// TIA Portal V17 export
// export: Created 2025-03-07T09:19:12.5870165Z, ExportSetting WithDefaults, DisplayName Totally Integrated Automation Portal, DisplayVersion V17 Update 8, DisplayName TIA Portal Openness, DisplayVersion V17 Update 8, DisplayName TIA Portal Version Control Interface, DisplayVersion V17, DisplayName SINAMICS Startdrive Advanced, DisplayVersion V17 SP2, DisplayName SINAMICS Startdrive G110M, G120, G120C, G120D, G120P, G115D, DisplayVersion V17 SP2, DisplayName SINAMICS Startdrive G130, G150, S120, S150, SINAMICS MV, S210, DisplayVersion V17 SP2, DisplayName STEP 7 Professional, DisplayVersion V17 Update 8, DisplayName SINUMERIK ONE STEP 7 Toolbox, DisplayVersion V17 Update 12, DisplayName SINUMERIK 840D sl STEP 7 Toolbox, DisplayVersion V17 Update 12, DisplayName STEP 7 Safety, DisplayVersion V17 Update 6, DisplayName WinCC Advanced, DisplayVersion V17 Update 8
FUNCTION "FC7210_PRODUCTION" : Void   // FC7210, LAD
{ S7_Optimized_Access := 'FALSE' }
AUTHOR : ETXETAR
VERSION : 1.0
// stored: AutoNumber false, IsIECCheckEnabled false, SetENOAutomatically false, UDAEnableTagReadback false
   VAR_TEMP
      UNIT_01_ENABLE_COUNT : Bool;   // UNIT 01 ENABLE COUNT
      UNIT_02_ENABLE_COUNT : Bool;   // UNIT 02 ENABLE COUNT
   END_VAR
   VAR_TEMP   // added for the SCL form of the ladder/FBD networks
      _w1 : Bool;
   END_VAR
BEGIN

REGION Network 1: UNIT 01 ENABLE COUNT / ENABLE FIXTURE 1 COUNT
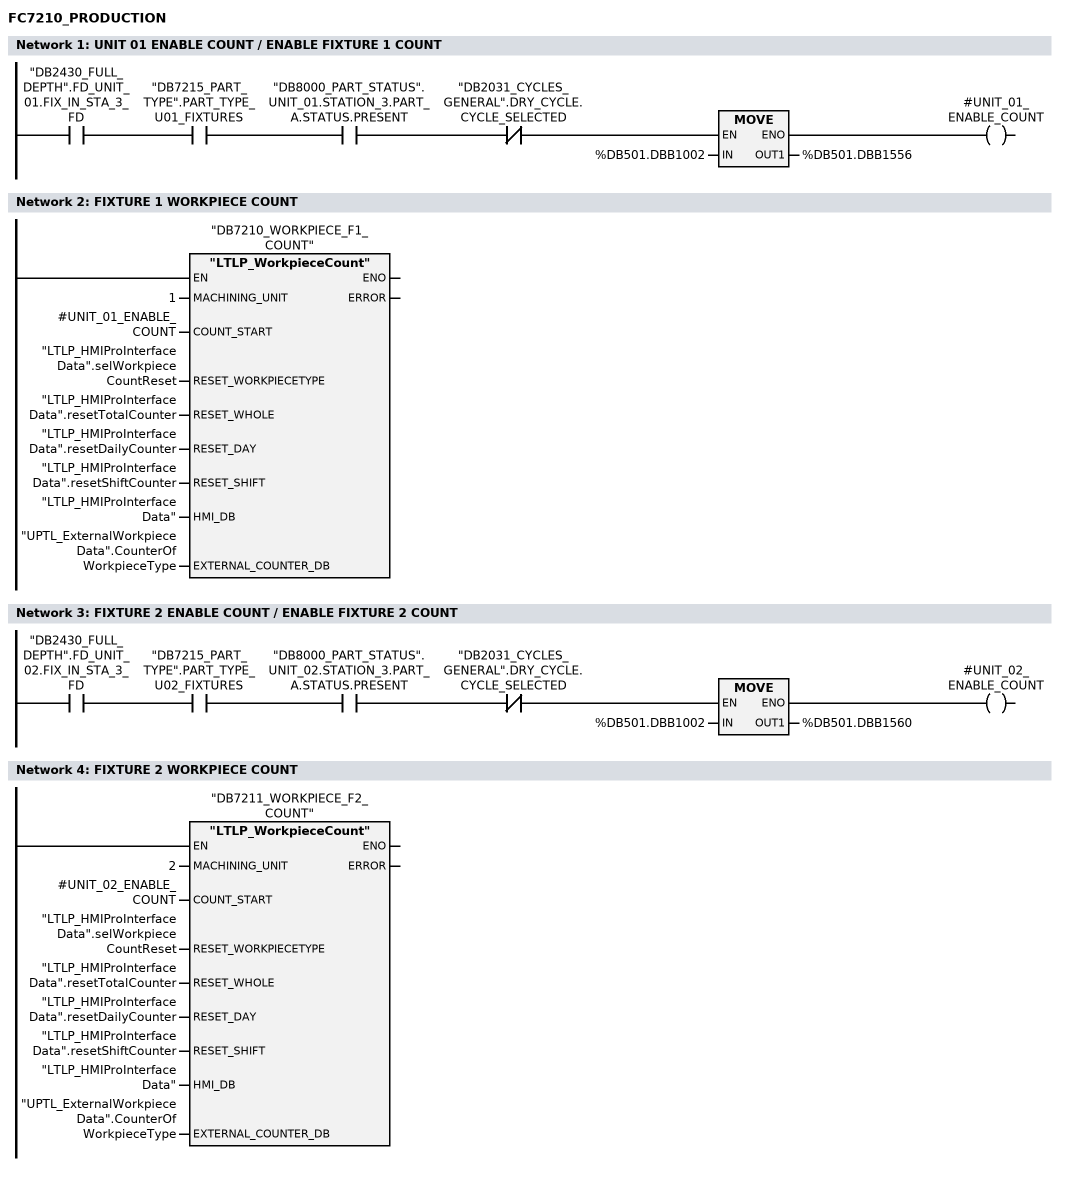
   RUNG wire#powerrail
      Contact( "DB2430_FULL_DEPTH".FD_UNIT_01.FIX_IN_STA_3_FD )
      Contact( "DB7215_PART_TYPE".PART_TYPE_U01_FIXTURES )
      Contact( "DB8000_PART_STATUS".UNIT_01.STATION_3.PART_A.STATUS.PRESENT )
      I_Contact( "DB2031_CYCLES_GENERAL".DRY_CYCLE.CYCLE_SELECTED )
      Move(in := %DB501.DBB1002, out1 => %DB501.DBB1556)
      Coil( #UNIT_01_ENABLE_COUNT )
   END_RUNG
   // the same network as SCL:
   #_w1 := "DB2430_FULL_DEPTH".FD_UNIT_01.FIX_IN_STA_3_FD AND "DB7215_PART_TYPE".PART_TYPE_U01_FIXTURES AND "DB8000_PART_STATUS".UNIT_01.STATION_3.PART_A.STATUS.PRESENT AND NOT "DB2031_CYCLES_GENERAL".DRY_CYCLE.CYCLE_SELECTED;
   IF #_w1 THEN %DB501.DBB1556 := %DB501.DBB1002; END_IF;
   #UNIT_01_ENABLE_COUNT := #_w1;
END_REGION

REGION Network 2: FIXTURE 1 WORKPIECE COUNT
   RUNG wire#powerrail
      "DB7210_WORKPIECE_F1_COUNT"(MACHINING_UNIT := 1, COUNT_START := #UNIT_01_ENABLE_COUNT, RESET_WORKPIECETYPE := "LTLP_HMIProInterfaceData".selWorkpieceCountReset, RESET_WHOLE := "LTLP_HMIProInterfaceData".resetTotalCounter, RESET_DAY := "LTLP_HMIProInterfaceData".resetDailyCounter, RESET_SHIFT := "LTLP_HMIProInterfaceData".resetShiftCounter, HMI_DB := "LTLP_HMIProInterfaceData", EXTERNAL_COUNTER_DB := "UPTL_ExternalWorkpieceData".CounterOfWorkpieceType, ERROR =>)
   END_RUNG
   // the same network as SCL:
   "DB7210_WORKPIECE_F1_COUNT"(MACHINING_UNIT := 1,   // "LTLP_WorkpieceCount"
                           COUNT_START := #UNIT_01_ENABLE_COUNT,
                           RESET_WORKPIECETYPE := "LTLP_HMIProInterfaceData".selWorkpieceCountReset,
                           RESET_WHOLE := "LTLP_HMIProInterfaceData".resetTotalCounter,
                           RESET_DAY := "LTLP_HMIProInterfaceData".resetDailyCounter,
                           RESET_SHIFT := "LTLP_HMIProInterfaceData".resetShiftCounter,
                           HMI_DB := "LTLP_HMIProInterfaceData",
                           EXTERNAL_COUNTER_DB := "UPTL_ExternalWorkpieceData".CounterOfWorkpieceType);
END_REGION

REGION Network 3: FIXTURE 2 ENABLE COUNT / ENABLE FIXTURE 2 COUNT
   RUNG wire#powerrail
      Contact( "DB2430_FULL_DEPTH".FD_UNIT_02.FIX_IN_STA_3_FD )
      Contact( "DB7215_PART_TYPE".PART_TYPE_U02_FIXTURES )
      Contact( "DB8000_PART_STATUS".UNIT_02.STATION_3.PART_A.STATUS.PRESENT )
      I_Contact( "DB2031_CYCLES_GENERAL".DRY_CYCLE.CYCLE_SELECTED )
      Move(in := %DB501.DBB1002, out1 => %DB501.DBB1560)
      Coil( #UNIT_02_ENABLE_COUNT )
   END_RUNG
   // the same network as SCL:
   #_w1 := "DB2430_FULL_DEPTH".FD_UNIT_02.FIX_IN_STA_3_FD AND "DB7215_PART_TYPE".PART_TYPE_U02_FIXTURES AND "DB8000_PART_STATUS".UNIT_02.STATION_3.PART_A.STATUS.PRESENT AND NOT "DB2031_CYCLES_GENERAL".DRY_CYCLE.CYCLE_SELECTED;
   IF #_w1 THEN %DB501.DBB1560 := %DB501.DBB1002; END_IF;
   #UNIT_02_ENABLE_COUNT := #_w1;
END_REGION

REGION Network 4: FIXTURE 2 WORKPIECE COUNT
   RUNG wire#powerrail
      "DB7211_WORKPIECE_F2_COUNT"(MACHINING_UNIT := 2, COUNT_START := #UNIT_02_ENABLE_COUNT, RESET_WORKPIECETYPE := "LTLP_HMIProInterfaceData".selWorkpieceCountReset, RESET_WHOLE := "LTLP_HMIProInterfaceData".resetTotalCounter, RESET_DAY := "LTLP_HMIProInterfaceData".resetDailyCounter, RESET_SHIFT := "LTLP_HMIProInterfaceData".resetShiftCounter, HMI_DB := "LTLP_HMIProInterfaceData", EXTERNAL_COUNTER_DB := "UPTL_ExternalWorkpieceData".CounterOfWorkpieceType, ERROR =>)
   END_RUNG
   // the same network as SCL:
   "DB7211_WORKPIECE_F2_COUNT"(MACHINING_UNIT := 2,   // "LTLP_WorkpieceCount"
                           COUNT_START := #UNIT_02_ENABLE_COUNT,
                           RESET_WORKPIECETYPE := "LTLP_HMIProInterfaceData".selWorkpieceCountReset,
                           RESET_WHOLE := "LTLP_HMIProInterfaceData".resetTotalCounter,
                           RESET_DAY := "LTLP_HMIProInterfaceData".resetDailyCounter,
                           RESET_SHIFT := "LTLP_HMIProInterfaceData".resetShiftCounter,
                           HMI_DB := "LTLP_HMIProInterfaceData",
                           EXTERNAL_COUNTER_DB := "UPTL_ExternalWorkpieceData".CounterOfWorkpieceType);
END_REGION
END_FUNCTION
